// TIA Portal V20 export
// export: Created 2026-04-11T06:02:30.7343802Z, ExportSetting WithDefaults, DisplayName Totally Integrated Automation Portal, DisplayVersion V20, DisplayName TIA Portal Openness, DisplayVersion V20, DisplayName TIA Portal Version Control Interface, DisplayVersion V20, DisplayName STEP 7 Professional, DisplayVersion V20, DisplayName STEP 7 Safety, DisplayVersion V20, DisplayName WinCC Basic/Comfort/Advanced, DisplayVersion V20, DisplayName WinCC Unified, DisplayVersion V20
TYPE "udtHandshake"
// stored: IsFailsafeCompliant false
   STRUCT
      bConnect { ExternalWritable := 'False'} : Bool;   // Connect request
      bRequest { ExternalWritable := 'False'} : Bool;   // Delivery request
      bRequestFast { ExternalWritable := 'False'} : Bool;   // Delivery fast request
      iQueue { ExternalWritable := 'False'} : Int;   // Number in queue
      iPriority { ExternalWritable := 'False'} : Int;   // Priority number, 0 = default
      rSetPoint { ExternalWritable := 'False'} : Real;   // Requested amount
   END_STRUCT;
END_TYPE
